(* CODESYS project ET3rdPartyDevices.library
   Version: 3.1.0.4
   Placeholder: ETX
   Description: Engineering Toolbox Extension Library for 3rd party devices
      
      The library is provided "as-is" for TwinCAT3.1 by the Beckhoff Industry Management for Electronics Manufacturing.
      The use of the Library is at the Customer's own risk
      Please check the "DisclaimerStatement" function of the EngineeringToolbox library >= v3.1.0.0
   Title: EngineeringToolboxExtension
   DefaultNamespace: ETX
   Company: Beckhoff Electronics Mfg

Project tree, tasks and I/O mapping:
  libraries: EngineeringToolbox, * (Beckhoff Electronics Mfg); Tc2_EtherCAT, * (Beckhoff Automation GmbH); Tc2_Standard, * (Beckhoff Automation GmbH); Tc2_System, * (Beckhoff Automation GmbH); Tc2_Utilities, * (Beckhoff Automation GmbH); Tc3_Module, * (Beckhoff Automation GmbH)
  GVLs/
  POUs/
    IO/
      Actuators/
        FreqConv/
          EtherCAT/
            DS402/
              Danfoss/
                function block CiA_DS402Controlword_Danfoss [ST]: createControlword
                function block CiA_DS402Statusword_Danfoss [ST]: readStatusword
                function block EcFcDS402_DanfossVLT302 [ST]: setDisable, setEnable, startForward, startReverse, switchOn, forwardStarted, isDisabled, isEnabled, isOff, isOn, reverseStarted
              Lenze/
                function block CiA_DS402Controlword_Lenze [ST]: createControlword
                function block CiA_DS402Statusword_Lenze [ST]: readStatusword
                function block EcFcDS402_LenzeI550 [ST]: setDisable, setEnable, startForward, startReverse, switchOn, forwardStarted, isDisabled, isEnabled, isOff, isOn, reverseStarted
              Parker/
                function block CiA_DS402Controlword_Parker [ST]: createControlword
                function block CiA_DS402Statusword_Parker [ST]: readStatusword
                function block EcFcDS402_ParkerAC30 [ST]: setDisable, setEnable, startForward, startReverse, switchOn, forwardStarted, isDisabled, isEnabled, isOff, isOn, reverseStarted
              Vacon/
                function block CiA_DS402Controlword_Vacon [ST]: createControlword
                function block CiA_DS402Statusword_Vacon [ST]: readStatusword
                function block EcFcDS402_VaconInd100 [ST]: setDisable, setEnable, startForward, startReverse, switchOn, forwardStarted, isDisabled, isEnabled, isOff, isOn, reverseStarted
            function block EcFcComSEW [ST]: reset, setContactorOFF, setContactorON, startBackward, startForward, switchOff, switchOn, backwardStarted, forwardStarted, inError, isBusy, isOff, isOn, noFeed, ok
        function block BlockEconomySmart [ST]: baseClock, reset
      Drives/
        CoE/
          InovanceSV660/
            function block AxDriveCoE_INOVNACE_wEvents [ST]
            function block CiA_DS402Statusword_INOVANCE [ST]: readStatusword
          StaeubliCS8/
            function block AxDriveCoE_StaeubliCS8 [ST]: confirm
            function block CiA_DS402Statusword_StaeubliCS8 [ST]: readStatusword
  VISUs/
*)

// POUs/IO/Actuators/FreqConv/EtherCAT/DS402/Danfoss/CiA_DS402Controlword_Danfoss
FUNCTION_BLOCK CiA_DS402Controlword_Danfoss EXTENDS CiA_DS402Controlword
VAR_INPUT
	EnableRamp						: BOOL; //Operation mode specific Bit 4 -> False = Quick stop / Switch on disabled  
	RunEnable						: BOOL;(* Operation mode specific Bit 5, False = Freeze, the given output frequency is maintained even iF the reference is changed. 
												TRUE = the frequency converter is again able to regulate, and the given reference is followed  *)
	Start							: BOOL;	(* Operation mode specific BIT 6 -> TRUE = gives a start command to the frequency converter / FALSE = the frequency converter controls the motor down to stop  *)

	Jog1On							: BOOL; //	Manufacturere specific Bit 11 Activation of pre-programmed speed in 8-90 Bus Jog 1 Speed JOG 1 is only possible if Bit 04="0", and bit 00-03="1". 

	SetupSelectLSB					: BOOL; //	Manufacturere specific Bit 13
		
	SetupSelectMSB					: BOOL; //	Manufacturere specific Bit 14
	Reversing						: BOOL; // Manufacturere specific Bit 15 
END_VAR
VAR_OUTPUT
END_VAR
VAR
END_VAR

;

METHOD PUBLIC createControlword : UINT
VAR_INPUT
	StatusState												: eCiA_DS402_STATUS_STATE;
END_VAR
	
	createControlword										:= SUPER^.createControlword(StatusState);
	createControlword.4										:= EnableRamp;
	createControlword.5										:= RunEnable;	
	createControlword.6										:= Start;	
	createControlword.11									:= Jog1On;	
	createControlword.13									:= SetupSelectLSB;	
	createControlword.14									:= SetupSelectMSB;	
	createControlword.15									:= Reversing;		
	
				
(*****************************************************************************)
END_METHOD

END_FUNCTION_BLOCK

// POUs/IO/Actuators/FreqConv/EtherCAT/DS402/Danfoss/CiA_DS402Statusword_Danfoss
FUNCTION_BLOCK CiA_DS402Statusword_Danfoss EXTENDS CiA_DS402Statusword
VAR_INPUT
END_VAR
VAR_OUTPUT	
	TargetReached				: BOOL; // Bit 10 in Velocity
	Running						: BOOL; //Bit 14
END_VAR

METHOD PUBLIC readStatusword : BOOL
VAR_INPUT
	Statusword 					:	UINT;
END_VAR


	TargetReached											:= Statusword.10;
	Running													:= Statusword.14;

	readStatusword											:= SUPER^.readStatusword(Statusword);
END_METHOD

END_FUNCTION_BLOCK

// POUs/IO/Actuators/FreqConv/EtherCAT/DS402/Danfoss/EcFcDS402_DanfossVLT302
{attribute 'no_check'}
// Control Danfoss frequency converter in FC mode
FUNCTION_BLOCK EcFcDS402_DanfossVLT302 EXTENDS EcFcDS402_ComBase IMPLEMENTS I_ActuatorFwdRev
VAR_INPUT
	VeloReference											: 	LREAL := 0.0;  	//[RPM] reference velocity
	RampUp													:	LREAL := 1.0;	//[s] sets slope of ramp
	RampDown												:	LREAL := 1.0;	//[s] sets slope of ramp
 
END_VAR                     							
VAR_OUTPUT                  							
	CiA_Control												:	CiA_DS402Controlword_Danfoss;
	CiA_Status												:	CiA_DS402Statusword_Danfoss;
	ErrorCode										AT  %I*	:	UDINT; 			//1690: see also Danfoss documentation
	OpHours											AT  %I* : 	UDINT;			//1500: Operating Hours
	ActPower												: 	LREAL;			//actual scaled Power of drive 
	ActVelo													: 	LREAL;			//actual scaled velocity of drive
	ActCurrent												: 	LREAL;			//actual current consumption of drive
	Q_TargetVelo									AT  %Q* : 	INT;			//1682: Frequence converter set value velocity
	Q_RampUp										AT  %Q* :	UDINT;			// 341: Frequence converter ramp time up
	Q_RampDown										AT  %Q* :	UDINT;			// 342: Frequence converter ramp time down 
END_VAR                 							
VAR (* IO Internal *)   							
                        							
	_ActVelo										AT  %I* : 	INT; 			//1605: Frequence converter actual velocity in digits based on VeloReference
	_ActCurrent										AT  %I* : 	DINT;			//1614: actual current consumption of drive
	_Power											AT  %I* : 	DINT;			//1610: Power 
END_VAR                 								
VAR                     	
END_VAR

(* Com Danfoss VLT302 over Ethercat Gateway MCA 124 	V1.0	 	*)
// ******************************************************************
{info 'FB EcFcDS402_DanfossVLT302: set parameter 4-10 to [2] both directions'}

(* Protection Switch *******************************************)		
	IF ResetTrig  
	THEN 
		REset(); 
	END_IF
	
	ProtSwitchOK();	
	FuseBreakOK(); (* same parameter like ProtSwitch *)

(* Contactor ***************************************************)
	Q_Contactor 											:= Contactor AND ProtSwitchOK.Q AND FuseBreakOK.Q;

(* Read status *************************************************)
	CiA_Status.readStatusword(Statusword);

(* interpret status word ***************************************)
	ActVelo													:= SCALE(_ActVelo, -16384, 16384, -VeloReference, VeloReference);	//16#F000 = -16384 | 16#4000 = 16384    
	ActCurrent             									:= TO_LREAL(_ActCurrent) / 100.0;
	ActPower												:= TO_LREAL(_Power) / 100.0;
	
	Ready													:= CiA_Status.ReadyToSwitchOn AND Q_Contactor;
	Error													:= CiA_Status.Fault AND Q_Contactor;                       									
	Busy													:= CiA_Status.OperationEnabled AND ActVelo <> 0; 
	                                        
// write contorlword DS 402  ****************************************
	CiA_Control.SwitchOn									:= Enable AND Q_Contactor;
	CiA_Control.EnableOperation								:= FeedBwd AND StartBwd AND NOT Start OR Feed AND Start AND NOT StartBwd;
	CiA_Control.FaultReset									:= ResetIntern;
	
	CiA_Control.EnableRamp			 						:= TRUE;
	CiA_Control.RunEnable									:= CiA_Control.SwitchOn;							       
	CiA_Control.Start										:= CiA_Control.EnableOperation;						                     	
	CiA_Control.Reversing			 						:= Start AND NOT StartBwd;	// 15 Reverse     
			
(* setvalue ***************************************************)
	IF CiA_Control.EnableOperation
	THEN
		Q_TargetVelo										:= TO_INT(SCALE(Velo, 	0, VeloReference, 0, 16384));
	ELSE
		Q_TargetVelo										:= 0;
	END_IF
	
	Q_RampUp 												:= TO_UDINT(RampUp*100);
	Q_RampDown 												:= TO_UDINT(RampDown*100);
	              
// Reset FALSE ****************************************************
	ResetIntern												:= FALSE;
	
(* HmiStatus **************************************************)
	Status.0 												:= CiA_Status.OperationEnabled AND StartBwd; 	// counter-clockwise rotation
	Status.1 												:= CiA_Status.OperationEnabled AND Start; 	// clockwise rotation
	Status.2 												:= ActVelo < 0;
	Status.3												:= ActVelo > 0;
	Status.4 												:= FeedBwd;
	Status.5 												:= Feed;
	Status.6 												:= Ready;
	Status.7 												:= Error;
// ****************************************************************

METHOD setDisable : BOOL
VAR_INPUT
END_VAR

SetDisable													:= Super^.setDisable() AND NOT CiA_Status.SwitchedOn;
END_METHOD

METHOD setEnable : BOOL
VAR_INPUT
END_VAR

SetEnable													:= SUPER^.setEnable() AND CiA_Status.SwitchedOn;
END_METHOD

METHOD PUBLIC startForward : bool //Return busy flag
VAR_INPUT
END_VAR
Start 														:= TRUE; 
StartBwd 													:= FALSE;
startForward												:= Busy and Q_TargetVelo > 0;
END_METHOD

METHOD PUBLIC startReverse : bool //Return busy flag
VAR_INPUT
END_VAR
Start 														:= FALSE; 
StartBwd 													:= TRUE;
startReverse												:= Busy and Q_TargetVelo < 0;
END_METHOD

METHOD PUBLIC switchOn : BOOL  //True if motor is switched on
VAR_INPUT
END_VAR
switchOn := startForward();
END_METHOD

{attribute 'monitoring' := 'call'}
PROPERTY public forwardStarted : BOOL
GET
forwardStarted := CiA_Control.EnableOperation and Q_TargetVelo > 0;
END_GET
END_PROPERTY

{attribute 'monitoring' := 'call'}
PROPERTY public isDisabled : BOOL
GET
isDisabled := not CiA_Status.SwitchedOn and not CiA_Status.OperationEnabled;
END_GET
END_PROPERTY

{attribute 'monitoring' := 'call'}
PROPERTY public isEnabled : BOOL
GET
isEnabled := CiA_Status.SwitchedOn or CiA_Status.OperationEnabled;
END_GET
END_PROPERTY

{attribute 'monitoring' := 'call'}
PROPERTY public isOff : BOOL
GET
isOff := NOT CiA_Status.OperationEnabled;
END_GET
END_PROPERTY

{attribute 'monitoring' := 'call'}
PROPERTY public isOn : BOOL
GET
isOn := CiA_Status.OperationEnabled;
END_GET
END_PROPERTY

{attribute 'monitoring' := 'call'}
PROPERTY public reverseStarted : BOOL
GET
reverseStarted := CiA_Control.EnableOperation and Q_TargetVelo < 0;
END_GET
END_PROPERTY

END_FUNCTION_BLOCK

// POUs/IO/Actuators/FreqConv/EtherCAT/DS402/Lenze/CiA_DS402Controlword_Lenze
FUNCTION_BLOCK CiA_DS402Controlword_Lenze EXTENDS CiA_DS402Controlword
VAR_INPUT
	Halt 					: BOOL; // Manufacturere specific Bit 8 - TRUE = stop motor
	ReleaseBreak			: BOOL; //Manufacturere specific Bit 14 
END_VAR
VAR_OUTPUT
END_VAR
VAR
END_VAR

;

METHOD PUBLIC createControlword : UINT
VAR_INPUT
	StatusState												: eCiA_DS402_STATUS_STATE;
END_VAR
	
	createControlword										:= SUPER^.createControlword(StatusState);
	createControlword.8										:= Halt;
	createControlword.8										:= ReleaseBreak;	
	
(*****************************************************************************)
END_METHOD

END_FUNCTION_BLOCK

// POUs/IO/Actuators/FreqConv/EtherCAT/DS402/Lenze/CiA_DS402Statusword_Lenze
FUNCTION_BLOCK CiA_DS402Statusword_Lenze EXTENDS CiA_DS402Statusword
VAR_INPUT
END_VAR
VAR_OUTPUT	
	RPDOsNotActive				:	 BOOL; //Manufacturer specific_Bit8	

	TargetReached				: BOOL; // Bit 10 in velocity 

	BreakOpened					: BOOL; //Manufacturer specific_Bit14
	StoNotActive				: BOOL; //Manufacturer specific_Bit15
END_VAR

METHOD PUBLIC readStatusword : BOOL
VAR_INPUT
	Statusword 					:	UINT;
END_VAR
	RPDOsNotActive											:= Statusword.8;

	TargetReached											:= Statusword.10;

	BreakOpened												:= Statusword.14;
	StoNotActive											:= Statusword.15;

	readStatusword											:= SUPER^.readStatusword(Statusword);
END_METHOD

END_FUNCTION_BLOCK

// POUs/IO/Actuators/FreqConv/EtherCAT/DS402/Lenze/EcFcDS402_LenzeI550
{attribute 'no_check'}
FUNCTION_BLOCK EcFcDS402_LenzeI550 EXTENDS EcFcDS402_ComBase IMPLEMENTS I_ActuatorFwdRev
VAR_INPUT
END_VAR                     							                 							
VAR_OUTPUT                  								
	ActVelo											AT  %I* : 	INT; 			//Actual velocity in rpm
	CiA_Control										:	CiA_DS402Controlword_Lenze;
	CiA_Status										:	CiA_DS402Statusword_Lenze;
	Q_TargetVelo								AT  %Q* : 	INT; 			//Set velocity in rpm
END_VAR                 							                 							
VAR    		
END_VAR

(* Com Lenze i550 over Ethercat Gateway 							*)
(********************************************************************)

(* Protection Switch *******************************************)		
	IF ResetTrig  
	THEN 
		REset(); 
	END_IF
	
	ProtSwitchOK();	
	FuseBreakOK(); (* same parameter like ProtSwitch *)

(* Contactor ***************************************************)
	Q_Contactor 											:= Contactor AND ProtSwitchOK.Q AND FuseBreakOK.Q;
	
(* Read status *************************************************)
	CiA_Status.readStatusword(Statusword);

(* interpret status word ***************************************)
	Ready													:= CiA_Status.ReadyToSwitchOn AND Q_Contactor;
	Error													:= CiA_Status.Fault AND Q_Contactor;                       									
	Busy													:= CiA_Status.OperationEnabled AND ActVelo <> 0; 
	                        	
(* write contorlword DS 402  **********************************)
	CiA_Control.SwitchOn									:= Enable AND Q_Contactor;
	CiA_Control.EnableOperation								:= FeedBwd AND StartBwd AND NOT Start OR Feed AND Start AND NOT StartBwd;
	CiA_Control.FaultReset									:= ResetIntern;	
	           									
(* setvalue ***************************************************)
	IF CiA_Control.EnableOperation
	THEN
		Q_TargetVelo										:= SEL(StartBwd, TO_INT(Velo), TO_INT(Velo) * -1);
	ELSE
		Q_TargetVelo										:= 0;
	END_IF

(* Write control word ******************************************)
	ControlWord 											:= CiA_Control.createControlword(CiA_Status.State);

(* Ack FALSE ***************************************************)
	ResetIntern												:= FALSE;
	
(* HmiStatus **************************************************)
	Status.0 												:= CiA_Status.OperationEnabled AND StartBwd; 	// counter-clockwise rotation
	Status.1 												:= CiA_Status.OperationEnabled AND Start; 	// clockwise rotation
	Status.2 												:= ActVelo < 0;
	Status.3												:= ActVelo > 0;
	Status.4 												:= FeedBwd;
	Status.5 												:= Feed;
	Status.6 												:= Ready;
	Status.7 												:= Error;
	                    									

(**************************************************************)

METHOD setDisable : BOOL
VAR_INPUT
END_VAR

SetDisable													:= Super^.setDisable() AND NOT CiA_Status.SwitchedOn;
END_METHOD

METHOD setEnable : BOOL
VAR_INPUT
END_VAR

SetEnable													:= SUPER^.setEnable() AND CiA_Status.SwitchedOn;
END_METHOD

METHOD PUBLIC startForward : bool //Return busy flag
VAR_INPUT
END_VAR
Start 														:= TRUE; 
StartBwd 													:= FALSE;
startForward												:= Busy and Q_TargetVelo > 0;
END_METHOD

METHOD PUBLIC startReverse : bool //Return busy flag
VAR_INPUT
END_VAR
Start 														:= FALSE; 
StartBwd 													:= TRUE;
startReverse												:= Busy and Q_TargetVelo < 0;
END_METHOD

METHOD PUBLIC switchOn : BOOL  //True if motor is switched on
VAR_INPUT
END_VAR
switchOn := startForward();
END_METHOD

{attribute 'monitoring' := 'call'}
PROPERTY public forwardStarted : BOOL
GET
forwardStarted := CiA_Control.EnableOperation and Q_TargetVelo > 0;
END_GET
END_PROPERTY

{attribute 'monitoring' := 'call'}
PROPERTY public isDisabled : BOOL
GET
isDisabled := not CiA_Status.SwitchedOn and not CiA_Status.OperationEnabled;
END_GET
END_PROPERTY

{attribute 'monitoring' := 'call'}
PROPERTY public isEnabled : BOOL
GET
isEnabled := CiA_Status.SwitchedOn or CiA_Status.OperationEnabled;
END_GET
END_PROPERTY

{attribute 'monitoring' := 'call'}
PROPERTY public isOff : BOOL
GET
isOff := NOT CiA_Status.OperationEnabled;
END_GET
END_PROPERTY

{attribute 'monitoring' := 'call'}
PROPERTY public isOn : BOOL
GET
isOn := CiA_Status.OperationEnabled;
END_GET
END_PROPERTY

{attribute 'monitoring' := 'call'}
PROPERTY public reverseStarted : BOOL
GET
reverseStarted := CiA_Control.EnableOperation and Q_TargetVelo < 0;
END_GET
END_PROPERTY

END_FUNCTION_BLOCK

// POUs/IO/Actuators/FreqConv/EtherCAT/DS402/Parker/CiA_DS402Controlword_Parker
FUNCTION_BLOCK CiA_DS402Controlword_Parker EXTENDS CiA_DS402Controlword
VAR_INPUT
	EnableRampOutput				: BOOL; //Operation mode specific Bit 4 - =0 to set ramp output to zero
	EnableRamp						: BOOL;	//Operation mode specific Bit 5 - =0 to hold ramp
	EnableRampInput					: BOOL;	//Operation mode specific Bit 6 - =0 to set ramp input to zero

	Jog1On							: BOOL; //	Manufacturere specific Bit 8 	

	AutoInitialise					: BOOL; //	Manufacturere specific Bit 12 - 1 = Allow SWITCH ON DISABLED to READY TO SWITCH ON transition regardless of bit 0 (Switch On)
	EnableRevOp						: BOOL; //	Manufacturere specific Bit 13 - 1 = Run Reverse
	RemoteCtrl						: BOOL; //	Manufacturere specific Bit 14 - 0 = Local Sequencing
	RemoteRef						: BOOL; //	Manufacturere specific Bit 15 - 0 = Local Reference
END_VAR
VAR_OUTPUT
END_VAR
VAR
END_VAR

;

METHOD PUBLIC createControlword : UINT
VAR_INPUT
	StatusState												: eCiA_DS402_STATUS_STATE;
END_VAR
	
	createControlword										:= SUPER^.createControlword(StatusState);
	createControlword.4										:= EnableRampOutput;
	createControlword.5										:= EnableRamp;	
	createControlword.6										:= EnableRampInput;	
	createControlword.12									:= AutoInitialise;	
	createControlword.13									:= EnableRevOp;	
	createControlword.14									:= RemoteCtrl;	
	createControlword.15									:= RemoteRef;		
	
(*****************************************************************************)
END_METHOD

END_FUNCTION_BLOCK

// POUs/IO/Actuators/FreqConv/EtherCAT/DS402/Parker/CiA_DS402Statusword_Parker
FUNCTION_BLOCK CiA_DS402Statusword_Parker EXTENDS CiA_DS402Statusword
VAR_INPUT
END_VAR
VAR_OUTPUT	
	TargetReached				: BOOL; // Bit 10 
	Running						: BOOL; //Bit 14
END_VAR

METHOD PUBLIC readStatusword : BOOL
VAR_INPUT
	Statusword 					:	UINT;
END_VAR


	TargetReached											:= Statusword.10;
	Running													:= Statusword.14;

	readStatusword											:= SUPER^.readStatusword(Statusword);
END_METHOD

END_FUNCTION_BLOCK

// POUs/IO/Actuators/FreqConv/EtherCAT/DS402/Parker/EcFcDS402_ParkerAC30
{attribute 'no_check'}
FUNCTION_BLOCK EcFcDS402_ParkerAC30 EXTENDS EcFcDS402_ComBase IMPLEMENTS I_ActuatorFwdRev
VAR_INPUT
	RefVelo													: 	LREAL := 2000; 	//sets speed of rotation	
	RampUp											AT  %Q*	:	TIME := T#10S;	//0486: Acceleration Time
	RampDown										AT  %Q*	:	TIME := T#10S;	//0487: Deceleration Time
END_VAR                     							
VAR_OUTPUT               
	CiA_Control												:	CiA_DS402Controlword_Parker;
	CiA_Status												:	CiA_DS402Statusword_Parker;

	{attribute 'displaymode':='hex'}   							
	WarningCode										AT  %I*	:	UDINT;			//0829: Warnings  1 - 32
	ActVelo											AT  %I* : 	REAL; 			//0395: Actual Speed Percent
	Power											AT  %I*	: 	REAL; 			//0380: Power kW
	Q_TargetVelo							 	AT  %Q* :	REAL;			//0681: Comms Reference
END_VAR                 							
VAR (* IO Internal *)   							
END_VAR                 								
VAR                     	
END_VAR

(* Com Parker AC30 										V1.0   *)
(***************************************************************)

(* Protection Switch *******************************************)		
	IF ResetTrig  
	THEN 
		REset(); 
	END_IF
	
	ProtSwitchOK();	
	FuseBreakOK(); (* same parameter like ProtSwitch *)

(* Contactor ***************************************************)
	Q_Contactor 											:= Contactor AND ProtSwitchOK.Q AND FuseBreakOK.Q;

(* Read status *************************************************)
	CiA_Status.readStatusword(Statusword);

(* interpret status word ***************************************)
	Ready													:= CiA_Status.ReadyToSwitchOn AND Q_Contactor;
	Error													:= CiA_Status.Fault AND Q_Contactor;                       									
	Busy													:= CiA_Status.OperationEnabled AND ActVelo <> 0; 
	                                        
// write contorlword DS 402  ****************************************
	CiA_Control.SwitchOn									:= Enable AND Q_Contactor;
	CiA_Control.EnableOperation								:= FeedBwd AND StartBwd AND NOT Start OR Feed AND Start AND NOT StartBwd;
	CiA_Control.FaultReset									:= ResetIntern;
	CiA_Control.EnableRevOp									:= CiA_Control.EnableOperation AND 	StartBwd;						

(* setvalue ***************************************************)
	IF CiA_Control.EnableOperation AND RefVelo <> 0.0
	THEN
		IF StartBwd
		THEN
			Q_TargetVelo 									:= TO_REAL(Velo/RefVelo * 100.0  * -1); (* 1 Digit = 1 rpm *)
		ELSE	
			Q_TargetVelo									:= TO_REAL(Velo/RefVelo * 100.0); (* 1 Digit = 1 rpm *)
		END_IF	
	ELSE
		Q_TargetVelo										:= 0;
	END_IF
	
// Reset FALSE ****************************************************
	ResetIntern												:= FALSE;
	
(* HmiStatus **************************************************)
	Status.0 												:= CiA_Status.OperationEnabled AND StartBwd; 	// counter-clockwise rotation
	Status.1 												:= CiA_Status.OperationEnabled AND Start; 	// clockwise rotation
	Status.2 												:= ActVelo < 0;
	Status.3												:= ActVelo > 0;
	Status.4 												:= FeedBwd;
	Status.5 												:= Feed;
	Status.6 												:= Ready;
	Status.7 												:= Error;
// ****************************************************************

METHOD setDisable : BOOL
VAR_INPUT
END_VAR

SetDisable													:= Super^.setDisable() AND NOT CiA_Status.SwitchedOn;
END_METHOD

METHOD setEnable : BOOL
VAR_INPUT
END_VAR

SetEnable													:= SUPER^.setEnable() AND CiA_Status.SwitchedOn;
END_METHOD

METHOD PUBLIC startForward : bool //Return busy flag
VAR_INPUT
END_VAR
Start 														:= TRUE; 
StartBwd 													:= FALSE;
startForward												:= Busy and Q_TargetVelo > 0;
END_METHOD

METHOD PUBLIC startReverse : bool //Return busy flag
VAR_INPUT
END_VAR
Start 														:= FALSE; 
StartBwd 													:= TRUE;
startReverse												:= Busy and Q_TargetVelo < 0;
END_METHOD

METHOD PUBLIC switchOn : BOOL  //True if motor is switched on
VAR_INPUT
END_VAR
switchOn := startForward();
END_METHOD

{attribute 'monitoring' := 'call'}
PROPERTY public forwardStarted : BOOL
GET
forwardStarted := CiA_Control.EnableOperation and Q_TargetVelo > 0;
END_GET
END_PROPERTY

{attribute 'monitoring' := 'call'}
PROPERTY public isDisabled : BOOL
GET
isDisabled := not CiA_Status.SwitchedOn and not CiA_Status.OperationEnabled;
END_GET
END_PROPERTY

{attribute 'monitoring' := 'call'}
PROPERTY public isEnabled : BOOL
GET
isEnabled := CiA_Status.SwitchedOn or CiA_Status.OperationEnabled;
END_GET
END_PROPERTY

{attribute 'monitoring' := 'call'}
PROPERTY public isOff : BOOL
GET
isOff := NOT CiA_Status.OperationEnabled;
END_GET
END_PROPERTY

{attribute 'monitoring' := 'call'}
PROPERTY public isOn : BOOL
GET
isOn := CiA_Status.OperationEnabled;
END_GET
END_PROPERTY

{attribute 'monitoring' := 'call'}
PROPERTY public reverseStarted : BOOL
GET
reverseStarted := CiA_Control.EnableOperation and Q_TargetVelo < 0;
END_GET
END_PROPERTY

END_FUNCTION_BLOCK

// POUs/IO/Actuators/FreqConv/EtherCAT/DS402/Vacon/CiA_DS402Controlword_Vacon
FUNCTION_BLOCK CiA_DS402Controlword_Vacon EXTENDS CiA_DS402Controlword
VAR_INPUT
	AlarmReset				:	BOOL; //Manufacturere specific Bit 12 

END_VAR
VAR_OUTPUT
END_VAR
VAR
END_VAR

;

METHOD PUBLIC createControlword : UINT
VAR_INPUT
	StatusState												: eCiA_DS402_STATUS_STATE;
END_VAR
	
	createControlword										:= SUPER^.createControlword(StatusState);
	createControlword.11									:= AlarmReset;	
	
(*****************************************************************************)
END_METHOD

END_FUNCTION_BLOCK

// POUs/IO/Actuators/FreqConv/EtherCAT/DS402/Vacon/CiA_DS402Statusword_Vacon
FUNCTION_BLOCK CiA_DS402Statusword_Vacon EXTENDS CiA_DS402Statusword
VAR_INPUT
END_VAR
VAR_OUTPUT	
	TargetReached				: BOOL; // Bit 10 commonly used FOR in target position, velocity ect.
	IncorrectDriveMode		:	BOOL; //Manufacturer specific_Bit14
END_VAR

METHOD PUBLIC readStatusword : BOOL
VAR_INPUT
	Statusword 					:	UINT;
END_VAR


	TargetReached											:= Statusword.10;

	IncorrectDriveMode										:= Statusword.14;


	readStatusword											:= SUPER^.readStatusword(Statusword);
END_METHOD

END_FUNCTION_BLOCK

// POUs/IO/Actuators/FreqConv/EtherCAT/DS402/Vacon/EcFcDS402_VaconInd100
{attribute 'no_check'}
FUNCTION_BLOCK EcFcDS402_VaconInd100 EXTENDS EcFcDS402_ComBase IMPLEMENTS I_ActuatorFwdRev
VAR_INPUT
END_VAR                     							
VAR_OUTPUT                  								
	CiA_Control										:	CiA_DS402Controlword_Vacon;
	CiA_Status										:	CiA_DS402Statusword_Vacon;
	_1_OutputFreq 							AT  %I*	:	UINT; // 0,01 Hz
	_2_Act_rpm								AT  %I*	:	UINT; // 1/MIN
	_3_ActCurrent							AT  %I*	:	UINT; // 0,1 A
	_4_ActTorque							AT  %I*	:	UINT; // 0.1%
	_5_ActPower								AT  %I*	:	UINT; // 0.1%
	_6_ActVoltage							AT  %I*	:	UINT; // 0,1 V
	_7_DClinkVoltage						AT  %I*	:	UINT; // 1 V
	_8_LastErrorCode						AT  %I*	:	UINT; //  
	Q_TargetVelo									AT  %Q* : 	INT; 			//Set velocity in rpm
END_VAR                 							
VAR (* IO Internal *)   							

END_VAR

(* Com Vacon 100 +SDEC EtherCAT Fieldbus option Board 	V1.0   *)
(***************************************************************)
																													
(* Protection Switch *******************************************)		
	IF ResetTrig  
	THEN 
		REset(); 
	END_IF
	
	ProtSwitchOK();	
	FuseBreakOK(); (* same parameter like ProtSwitch *)

(* Contactor ***************************************************)
	Q_Contactor 											:= Contactor AND ProtSwitchOK.Q AND FuseBreakOK.Q;
	
(* Read status *************************************************)
	CiA_Status.readStatusword(Statusword);

(* interpret status word ***************************************)
	Ready													:= CiA_Status.ReadyToSwitchOn AND Q_Contactor;
	Error													:= CiA_Status.Fault AND Q_Contactor;                       									
	Busy													:= CiA_Status.OperationEnabled AND _2_Act_rpm <> 0; 
	                        	
(* write contorlword DS 402  **********************************)
	CiA_Control.SwitchOn									:= Enable AND Q_Contactor;
	CiA_Control.EnableOperation								:= FeedBwd AND StartBwd AND NOT Start OR Feed AND Start AND NOT StartBwd;
	CiA_Control.FaultReset									:= ResetIntern;	
	CiA_Control.AlarmReset									:= ResetIntern;	
	           									
(* setvalue ***************************************************)
	IF CiA_Control.EnableOperation
	THEN
		Q_TargetVelo										:= SEL(StartBwd, TO_INT(Velo), TO_INT(Velo) * -1);
	ELSE
		Q_TargetVelo										:= 0;
	END_IF

(* Write control word ******************************************)
	ControlWord 											:= CiA_Control.createControlword(CiA_Status.State);

(* Ack FALSE ***************************************************)
	ResetIntern												:= FALSE;
	
(* HmiStatus **************************************************)
	Status.0 												:= CiA_Status.OperationEnabled AND StartBwd; 	// counter-clockwise rotation
	Status.1 												:= CiA_Status.OperationEnabled AND Start; 	// clockwise rotation
	Status.2 												:= _2_Act_rpm < 0;
	Status.3												:= _2_Act_rpm > 0;
	Status.4 												:= FeedBwd;
	Status.5 												:= Feed;
	Status.6 												:= Ready;
	Status.7 												:= Error;
	                    									

(**************************************************************)

METHOD setDisable : BOOL
VAR_INPUT
END_VAR

SetDisable													:= Super^.setDisable() AND NOT CiA_Status.SwitchedOn;
END_METHOD

METHOD setEnable : BOOL
VAR_INPUT
END_VAR

SetEnable													:= SUPER^.setEnable() AND CiA_Status.SwitchedOn;
END_METHOD

METHOD PUBLIC startForward : bool //Return busy flag
VAR_INPUT
END_VAR
Start 														:= TRUE; 
StartBwd 													:= FALSE;
startForward												:= Busy and Q_TargetVelo > 0;
END_METHOD

METHOD PUBLIC startReverse : bool //Return busy flag
VAR_INPUT
END_VAR
Start 														:= FALSE; 
StartBwd 													:= TRUE;
startReverse												:= Busy and Q_TargetVelo < 0;
END_METHOD

METHOD PUBLIC switchOn : BOOL  //True if motor is switched on
VAR_INPUT
END_VAR
switchOn := startForward();
END_METHOD

{attribute 'monitoring' := 'call'}
PROPERTY public forwardStarted : BOOL
GET
forwardStarted := CiA_Control.EnableOperation and Q_TargetVelo > 0;
END_GET
END_PROPERTY

{attribute 'monitoring' := 'call'}
PROPERTY public isDisabled : BOOL
GET
isDisabled := not CiA_Status.SwitchedOn and not CiA_Status.OperationEnabled;
END_GET
END_PROPERTY

{attribute 'monitoring' := 'call'}
PROPERTY public isEnabled : BOOL
GET
isEnabled := CiA_Status.SwitchedOn or CiA_Status.OperationEnabled;
END_GET
END_PROPERTY

{attribute 'monitoring' := 'call'}
PROPERTY public isOff : BOOL
GET
isOff := NOT CiA_Status.OperationEnabled;
END_GET
END_PROPERTY

{attribute 'monitoring' := 'call'}
PROPERTY public isOn : BOOL
GET
isOn := CiA_Status.OperationEnabled;
END_GET
END_PROPERTY

{attribute 'monitoring' := 'call'}
PROPERTY public reverseStarted : BOOL
GET
reverseStarted := CiA_Control.EnableOperation and Q_TargetVelo < 0;
END_GET
END_PROPERTY

END_FUNCTION_BLOCK

// POUs/IO/Actuators/FreqConv/EtherCAT/EcFcComSEW
{attribute 'no_check'}
FUNCTION_BLOCK EcFcComSEW IMPLEMENTS I_ActuatorFwdBwd(* SEW *)
VAR_INPUT
	ResetTrig												:	BOOL := TRUE;	//Resets error with rising edge 
	Start													:	BOOL := FALSE;	//motor rotates in right direction when TRUE
	StartBwd												:	BOOL := FALSE; 	//motor rotates in left direction when TRUE
	Contactor												:	BOOL := FALSE;	//if available
	Enable													:	BOOL := FALSE;	//enables drive
	Feed													:	BOOL := TRUE;	//enables feed in right direction and should be set to FALSE when right limit sensor is reached
	FeedBwd													:	BOOL := TRUE;	//enables feed in left direction and should be set to FALSE when left limit sensor is reached
	Velo													: 	LREAL := 0.0;  	//sets speed of rotation
	Ramp													:	LREAL := 1.0;	//sets slope of ramp
	ProtSwitchOK											: 	FUSE;			//monitors feeding protective device
	FuseBreakOK												: 	FUSE;			//monitors feeding circuit breaker 
END_VAR                     							
VAR_OUTPUT                  							
{attribute 'displaymode':='binary'}
	Status													:	BYTE; 			//for HMI
{attribute 'displaymode':='binary'}
	UnitStatus												:	BYTE; 			(* device status
																				0x0 not ready
																				0x1 controller locked
																				0x2 not enabled
																				0x3 standstill current acitve, not enabled
																				0x4 enabled
																				0x8 default factory settings active *)
	ErrorCode												:	BYTE; 			//see also SEW-documentation
{attribute 'displaymode':='hex'}
	Statusword1										AT  %I* : 	INT;			//status word 1 contains state of drive
	ActVelo													: 	LREAL;			//actual scaled velocity of drive
	ActCurrent										AT  %I* : 	INT;			//actual current consumption of drive
	Ready													:	BOOL;			//TRUE when drive is ready to operate
	Warning													:	BOOL;			//TRUE when a warning is active 
	Busy													:	BOOL;			//Busy is TRUE at the rising edge of Enable and stays TRUE as long as the FB is performing any action. 	
	Error													:	BOOL;			//Rising edge of Error informs that an error occurred during the execution of the Function Block 	 	
END_VAR                 							
VAR (* IO Internal *)
{attribute 'displaymode':='hex'}   							
	Q_Controlword1									AT  %Q* : 	INT;			//Frequence converter controlword 1
	Q_TargetVelo									AT  %Q* : 	INT;			//Frequence converter set target velocity in digits
	Q_Ramp											AT  %Q* :	INT;			//Frequence converter ramp time in 
                        							
	Q_Contactor 									AT  %Q* :	BOOL;			//Hardware output 
	_ActVeloDigit									AT  %I* : 	INT; 			//Frequence converter actual velocity in digits based on rpm 
END_VAR                 								
VAR    
	QuitIntern												:	BOOL;                 	
END_VAR

(* Com SEW MovitracB over Ethercat Gateway 		V2.0	*)
(********************************************************)

(* Protection Switch *****************************************)
	IF ResetTrig 
	THEN 
		reset(); 
	END_IF
	
	ProtSwitchOK();
	FuseBreakOK(); (* same parameter like ProtSwitch *)

(* Contactor ********************************************************)
	Q_Contactor 											:= Contactor AND ProtSwitchOK.Q AND FuseBreakOK.Q;

(* interpret status word *********************************)
	(*EndstufeFRG											:= Statusword1.0; *)
	Ready													:= Statusword1.1 AND Q_Contactor;
	Warning													:= Statusword1.5 AND Ready ;
	Error													:= Statusword1.5 AND NOT Ready AND Q_Contactor ;
	(*EndlLinksAktiv 										:= Statusword1.6; *)
	(*EndlLinksAktiv 										:= Statusword1.7; *)
                        									
	ActVelo													:= INT_TO_LREAL(_ActVeloDigit) * 0.2;
	Busy													:= Ready AND Q_Controlword1.2 AND ActVelo > 5.0;
                        	
(* interpret HighByte status word 1 ********************)
	(* Init *)
	UnitStatus := ErrorCode 								:= 0;

	IF Q_Contactor THEN
		IF NOT Statusword1.5 THEN
			UnitStatus.0 									:= Statusword1.8;
			UnitStatus.1 									:= Statusword1.9;
			UnitStatus.2 									:= Statusword1.10;
			UnitStatus.3									:= Statusword1.11;
			UnitStatus.4 									:= Statusword1.12;
			UnitStatus.5 									:= Statusword1.13;
			UnitStatus.6 									:= Statusword1.14;
			UnitStatus.7 									:= Statusword1.15;
		ELSE                								
			ErrorCode.0 									:= Statusword1.8;
			ErrorCode.1 									:= Statusword1.9;
			ErrorCode.2 									:= Statusword1.10;
			ErrorCode.3										:= Statusword1.11;
			ErrorCode.4 									:= Statusword1.12;
			ErrorCode.5 									:= Statusword1.13;
			ErrorCode.6 									:= Statusword1.14;
			ErrorCode.7 									:= Statusword1.15;
		END_IF
	END_IF

(* write contorlword 1  *********************************)
	Q_Controlword1.0 										:= FALSE; (* controller locked=1/0=enabled *)
	Q_Controlword1.1 										:= Enable AND Q_Contactor; (* controller enabled=1/0=rapid stop *)
	Q_Controlword1.2 										:= FeedBwd AND StartBwd AND NOT Start
																OR Feed AND Start AND NOT StartBwd; (* enable start FU *)
	Q_Controlword1.6 										:= QuitIntern;
	Q_Controlword1.8 										:= NOT Start AND StartBwd; (* rotation direction 0=right/1=left *)
                        									
(* setvalue **************************************)
	IF 	Start 
		AND NOT StartBwd 
		AND Feed 
	THEN
		Q_TargetVelo 										:= LREAL_TO_INT(Velo) * 5; (* 5 Digit = 1 rpm *)
	ELSIF StartBwd 
		AND NOT Start 
		AND FeedBwd 
	THEN
		Q_TargetVelo 										:= (LREAL_TO_INT(Velo) * 5 ) * -1; (* 5 Digit = 1 rpm *)
	ELSE
		Q_TargetVelo 										:= 0;
	END_IF

(* set ramp ******************************************)
	Q_Ramp	 												:= LREAL_TO_INT(Ramp);

(* Ack FALSE **********************************************)
	QuitIntern												:= FALSE;
	
(* HmiStatus **************************************************)
	Status.0 												:= Q_Controlword1.2 AND Q_Controlword1.8 ; //counter-clockwise rotation
	Status.1 												:= Q_Controlword1.2 AND NOT  Q_Controlword1.8; //clockwise rotation
	Status.2 												:= FALSE;
	Status.3												:= FALSE;
	Status.4 												:= FeedBwd;
	Status.5 												:= Feed;
	Status.7 												:= Ready;
	Status.7 												:= Error;
	                    									

(**************************************************************)

METHOD PUBLIC reset : booL
VAR_INPUT
END_VAR
QuitIntern 	:= Q_Controlword1.6   							:= TRUE;
ProtSwitchOK.reset();
FuseBreakOK.reset();
reset													:= TRUE;
END_METHOD

METHOD PUBLIC setContactorOFF : BOOL //Return true if contactor is off and not busy
VAR_INPUT
END_VAR
Q_Contactor := Contactor 									:=FALSE;
							
SetContactorOFF 											:= TRUE;
END_METHOD

METHOD PUBLIC setContactorON : bool //return true if contactor on
VAR_INPUT
END_VAR
Q_Contactor := Contactor 									:= ProtSwitchOK.Q AND FuseBreakOK.Q ;
SetContactorON												:= Q_Contactor;
END_METHOD

METHOD PUBLIC startBackward : bool //Return busy flag
VAR_INPUT
END_VAR
Start 														:= FALSE; 
StartBwd 													:= TRUE;
Q_Controlword1.2 											:= FeedBwd AND ProtSwitchOK.Q; (* FRG Start FU *)
Q_Controlword1.8 											:= Q_Controlword1.2 ; (* Drehrichtung 0=Rechts/1=Links *)
Busy														:= Q_Controlword1.2;
startBackward												:= Busy;
END_METHOD

METHOD PUBLIC startForward : bool //Return busy flag
VAR_INPUT
END_VAR
Start 														:= TRUE; 
StartBwd 													:= FALSE;
Q_Controlword1.2 											:= Feed AND Start AND NOT StartBwd AND ProtSwitchOK.Q; (* FRG Start FU *)
Q_Controlword1.8 											:= FALSE ; (* Drehrichtung 0=Rechts/1=Links *)
Busy														:= Q_Controlword1.2;
startForward												:= Busy;
END_METHOD

METHOD PUBLIC switchOff : BOOL //Return true if stopped / busy = false
VAR_INPUT
END_VAR
Start 														:= FALSE;
StartBwd													:= FALSE;
Q_Controlword1.2 											:= FALSE;
switchOff													:= NOT Busy;
END_METHOD

METHOD PUBLIC switchOn : BOOL  //True if motor is switched on
VAR_INPUT
END_VAR
switchOn := startForward();
END_METHOD

{attribute 'monitoring' := 'call'}
PROPERTY public backwardStarted : BOOL
GET
backwardStarted := Q_Controlword1.2 and Q_TargetVelo < 0;
END_GET
END_PROPERTY

{attribute 'monitoring' := 'call'}
PROPERTY public forwardStarted : BOOL
GET
forwardStarted := Q_Controlword1.2 and Q_TargetVelo > 0;
END_GET
END_PROPERTY

{attribute 'monitoring' := 'call'}
PROPERTY public inError : bool
GET
inError := Error or not ProtSwitchOK.Q or not FuseBreakOK.Q;
END_GET
END_PROPERTY

{attribute 'monitoring' := 'call'}
PROPERTY public isBusy : bool
GET
isBusy := Busy;
END_GET
END_PROPERTY

{attribute 'monitoring' := 'call'}
PROPERTY public isOff : BOOL
GET
isOff := NOT Q_Contactor or Q_TargetVelo = 0;
END_GET
END_PROPERTY

{attribute 'monitoring' := 'call'}
PROPERTY public isOn : BOOL
GET
isOn := Q_Contactor and Q_TargetVelo <> 0 and not inError;
END_GET
END_PROPERTY

{attribute 'monitoring' := 'call'}
PROPERTY noFeed : BOOL
GET
noFeed := NOT Feed and not FeedBwd;
END_GET
END_PROPERTY

{attribute 'monitoring' := 'call'}
PROPERTY ok : bool
GET
ok := isOn;
END_GET
END_PROPERTY

END_FUNCTION_BLOCK

// POUs/IO/Actuators/BlockEconomySmart
//Block Economy Smart 
//FB is able to control and read all values from Block Ecomemy Smart Fuse
{attribute 'no_check'}
FUNCTION_BLOCK BlockEconomySmart
VAR CONSTANT 										
	MIN_DATA												: INT := 0;
	MAX_DATA												: INT := 96;
END_VAR
VAR_OUTPUT CONSTANT
	MIN_CHANNEL												: INT := 1;
	MAX_CHANNEL												: INT := 8;
	STATUS_ON												: BYTE := 0;
	STATUS_OFF												: BYTE := 1;
	STATUS_TRIP												: BYTE := 2;
	STATUS_OVERCURRENT										: BYTE := 3;
END_VAR                         							
VAR_INPUT                       							
	Enable													: BOOL := TRUE; //Enable communication 
	Force													: ARRAY[MIN_CHANNEL..MAX_CHANNEL] OF BOOL; 	// 	simulates channel
	Control													: ARRAY[MIN_CHANNEL..MAX_CHANNEL] OF BOOL; 	// 	Enable/Disable channel 
	SetCtrl													: BOOL := FALSE;		// 	Write channel control to output (Econemy Smart Fuse)
	ResetTrig												: BOOL := FALSE;		// 	Reset tripped fuses/channels
	ReadSetValues											: BOOL := FALSE;		// 	Read trip set value of all cannels
	ReadChecksum											: BOOL := FALSE;		// 	Read checksumm
	ExtProtocolSampleingDivider								: UINT := 0;			//  0 = read only short protocol / >0 = read long protocol every n cycles 					
END_VAR
VAR_OUTPUT
	Voltage													: LREAL;					// [V] actual voltage
	Current													: ARRAY[MIN_CHANNEL..MAX_CHANNEL] OF LREAL;	// [A] actual cannel current[1-8]
	Status													: ARRAY[MIN_CHANNEL..MAX_CHANNEL] OF BYTE;	// Fuse status
	FuseTripped												: BOOL := FALSE;		// min 1 Fuse has tripped
	UpdateCycle												: UINT := 0;			// update Cycle counter
	Busy													: BOOL; 				// 
	ErrorCom												: BOOL;					// 				
END_VAR
VAR 
	In												AT%I*	: BOOL;
	Out												AT%Q*	: BOOL;
END_VAR
VAR
//local cache ************************************************************************************
	State													: INT := -1;
	CycleTime												: LREAL; // [ms] Cycle Time of PLC Task
	_BaseClock												: INT := 100; // MIN: 70 MAX: 200
	CurrentCycles											: UDINT;
	CyclePerTick											: UDINT;
	_InternReset											: BOOL;

	BitIdx,RecBits											: INT;
	SendData												: ARRAY[MIN_DATA..MAX_DATA] OF BOOL;
	ReceiveBits												: ARRAY[MIN_DATA..MAX_DATA] OF BOOL;
	ReceiveBytes											: ARRAY[MIN_DATA..MAX_DATA/8] OF BYTE;
	
	{attribute 'displaymode':='binary'}
	Temp 													: BYTE;		


				
//trigger *********************************************************************************
	
//timer ***********************************************************************************
	Delay													: TON;
	
//instances ***********************************************************************************             								
	GETCURTASKINDEX											: GETCURTASKINDEX;


//Dummys ****************************************************************************************
	i,j														: INT;
END_VAR

	(* Block Economy Smart communication 					*)
	(********************************************************)

(* Initiat reset of channel ***********************************************)
	IF ResetTrig THEN reset();	END_IF

(* State machine to read and write data ************************************)
	CASE State OF
	-1: // init
		GETCURTASKINDEX();
		CycleTime 											:= TwinCAT_SystemInfoVarList._TaskInfo[GETCURTASKINDEX.index].CycleTime / 10_000;
		IF CycleTime > 0 THEN           						
			CyclePerTick									:= LREAL_TO_UDINT(_BaseClock / CycleTime);	
			CyclePerTick									:= CyclePerTick + (CyclePerTick MOD 2);
			State											:= 0;
		END_IF                          						
																
	0: // idle          
		IF Enable
		THEN    	   
			Busy											:= TRUE; 						
			FOR i := MIN_CHANNEL TO MAX_CHANNEL DO    									
				SendData[i]									:= Control[9-i];
			END_FOR                 						
			SendData[9]										:= SetCtrl;			    	
			SendData[10]									:= extProtocolSampleingDivider <> 0
																AND(	
																(UpdateCycle MOD extProtocolSampleingDivider) = 0
																OR UpdateCycle = 0)
																OR ReadSetValues;
			SendData[11]									:= ReadSetValues;
			SendData[12]									:= FALSE;
			SendData[13]									:= FALSE;
			SendData[14]									:= ReadChecksum AND NOT SetCtrl;
			BitIdx											:= 0;		
			State											:= SEL(_InternReset, 10, 5); // Reset tripped if flag is true
			RecBits											:= SEL( SendData[10], 16, 88) 	// short / long
															+  SEL( ReadChecksum, 0, 8);	// checksum on/off
		ELSE
			Busy											:= FALSE;
			Out												:= FALSE;
			State											:= 0;
			Voltage											:= 0.0;
			MEMSET(ADR(Current),0,SIZEOF(Current));			
			MEMSET(ADR(Status),0,SIZEOF(Status));	        
			FuseTripped										:= FALSE;
			UpdateCycle										:= 0;		
		END_IF
																
	5:	//reset triped          								
		Out													:= TRUE;
		Delay(IN:= NOT Delay.Q, PT := T#600MS);             
															
		IF Delay.Q THEN             						
			_InternReset									:= FALSE;
			Delay(IN := FALSE);                             
			State 											:= 20;
		END_IF                  							
															
	10: // receive	            							
		Out													:= SendData[BitIdx] XOR CurrentCycles <= CyclePerTick / 2;		
															
		IF CurrentCycles >= CyclePerTick					 
		THEN                            	                
			ReceiveBits[BitIdx]								:= In;
			CurrentCycles									:= 0;
			BitIdx											:= BitIdx + 1;
			IF BitIdx > RecBits
			THEN
				Out											:= FALSE;
				State										:= 20;
			END_IF                  	
		ELSE	                    	
			CurrentCycles									:= CurrentCycles + 1;
		END_IF
		
	20:	 // interpret Channels
		Delay( IN:= NOT Delay.Q AND NOT IN, PT := TO_TIME(_BaseClock*3));
		IF Delay.Q THEN		// stop Bit		
			Delay(IN := FALSE);
			
			// Cannel Status
			FOR i := MIN_CHANNEL TO MAX_CHANNEL DO	
				IF Force[i] THEN
					Status[i]								:= STATUS_ON;				
				ELSIF ReceiveBits[9-i] AND ReceiveBits[17-i] THEN   
					Status[i]								:= STATUS_OVERCURRENT;	
				ELSIF ReceiveBits[9-i] THEN                     
					Status[i]								:= STATUS_ON;
				ELSIF ReceiveBits[17-i] THEN                    
					Status[i]								:= STATUS_TRIP;
				ELSE                                        
					Status[i]								:= STATUS_OFF;
				END_IF                                      
			END_FOR		                                    
		      
			//  interpret Checksum
			FOR i := MIN_DATA TO MAX_DATA/8 DO
				ReceiveBytes[0+i].0 						:= ReceiveBits[8*i+0];
				ReceiveBytes[0+i].1 						:= ReceiveBits[8*i+1];
				ReceiveBytes[0+i].2 						:= ReceiveBits[8*i+2];
				ReceiveBytes[0+i].3 						:= ReceiveBits[8*i+3];
				ReceiveBytes[0+i].4 						:= ReceiveBits[8*i+4];
				ReceiveBytes[0+i].5 						:= ReceiveBits[8*i+5];
				ReceiveBytes[0+i].6 						:= ReceiveBits[8*i+6];
				ReceiveBytes[0+i].7 						:= ReceiveBits[8*i+7];
			END_FOR
			ErrorCom := 	SendData[14]
						AND (	( ReceiveBytes[1] XOR ReceiveBytes[2]) = ReceiveBytes[3] AND BitIdx < 30
							OR 	((ReceiveBytes[1] XOR ReceiveBytes[2] XOR ReceiveBytes[3] XOR ReceiveBytes[4] XOR ReceiveBytes[5] XOR ReceiveBytes[6] XOR
						 		  ReceiveBytes[7] XOR ReceiveBytes[8] XOR ReceiveBytes[9] XOR ReceiveBytes[10] XOR ReceiveBytes[11]) = ReceiveBytes[12] AND BitIdx > 30)
							 );
                                              
			// set collective triped bit                    
			FuseTripped										:= FALSE;
			FOR i := MIN_CHANNEL TO MAX_CHANNEL DO          
				IF Status[i] = STATUS_TRIP THEN             
					FuseTripped								:= TRUE;
					EXIT;
				END_IF
			END_FOR
			
			// interpret extended protoccol
			IF 	SendData[10] 
				OR 	SendData[11] 
			THEN			
				FOR i := MIN_CHANNEL TO MAX_CHANNEL DO // Voltage
					Temp									:= SHL(Temp,1) OR TO_BYTE(ReceiveBits[16+i]);
				END_FOR		  
				Voltage										:= Temp/16.0 + 16;
				FOR j := MIN_CHANNEL TO MAX_CHANNEL DO // Current[1-8]
					FOR i := MIN_CHANNEL TO MAX_CHANNEL DO    // bit shifting
						Temp								:= SHL(Temp,1) OR TO_BYTE(ReceiveBits[24+((j-1)*8)+i]);
					END_FOR		  
					Current[j]								:= Temp/16.0;
				END_FOR
			END_IF          
				
			UpdateCycle 									:= UpdateCycle + 1; 
			State 											:= 0;
		END_IF	
	END_CASE
	
(*****************************************************************)

PROPERTY PUBLIC baseClock : INT // MIN: 70 MAX: 200
GET
BaseClock := _BaseClock;
END_GET
SET
_BaseClock := LIMIT(70, BaseClock, 200);
State := -1;
END_SET
END_PROPERTY

METHOD reset : BOOL //Resetting tripped channel / Return TRUE as lons as FuseTripped = TRUE
VAR_INPUT
END_VAR
_InternReset													:= FuseTripped;
reset															:= TRUE;
END_METHOD

END_FUNCTION_BLOCK

// POUs/IO/Drives/CoE/InovanceSV660/AxDriveCoE_INOVNACE_wEvents
FUNCTION_BLOCK AxDriveCoE_INOVNACE_wEvents  EXTENDS AxDriveBase (* Inovance SV660N EtherCAT drive 
Do enable remote break control the folloing settings are needed

Required process data: 
- 0x1B01, which includes 0x60FE:01 Physical outputs

Required startup list entries: 
- 0x60FE:02 (Bit Mask) = 400000 dec.
- 0x200D:12 (Forced DI/DO setting) = 4 dec (EtherCAT)
- 0x2004:05 (DO Function Selection) = 9 dec (to set DO function back to drive on restart) 

*)
VAR CONSTANT
	PHY_OUTPUT_BRAKE										:	INT := 18;
END_VAR
VAR_INPUT
	EnableEvent												:	BOOL := TRUE;
	ConfirmTrig												:	BOOL := FALSE; (* Reset event *)
	SourceId												:	UDINT := 102200; //CoE Drive default multisource Id + Ax id
	Name													:	STRING(30) := '';
	ErrorLimitPos											:	BOOL := FALSE;
	ErrorLimitNeg											:	BOOL := FALSE;
	BrakeUnlock												:	BOOL := FALSE;
	PhysicalOutputs									AT%Q*	:   UDINT;
END_VAR
VAR_OUTPUT
	BrakeUnlocked											:	BOOL;
	Status													:	CiA_DS402Statusword_INOVANCE;	

	EventStatus												:	DWORD;
	NoOfActiveEvents										:	INT;
	Busy													:	BOOL;
	Error													:	BOOL;
	ErrorId													:	UDINT;
	STOOff													:	BOOL;
	
	ModesOfOperationDisplay							AT %I*	:	SINT;
	DigitalInputs									AT %I*	:	UDINT;
	ErrorCode										AT %I*	:	UINT;
END_VAR
VAR
END_VAR
VAR
(* Function blocks ****************************************************************************)	
	CoEWrite												: FB_EcCoeSdoWriteEx := (tTimeout := DEFAULT_ADS_TIMEOUT);
	Event													: EventHandlingGrp10;
	i														:	INT;
	BrakeState												:	INT;	
	CoESetValue												:	INT;
END_VAR

	(* CoE Drive																		*)
	(************************************************************************************)

		(* CoE Drive																		*)
	(************************************************************************************)

(* abort function-call if the reference is invalid *****************************)
	IF NOT __ISVALIDREF(rAxis) 
	THEN
		Busy												:= NOT Error;
		Fault												:= TRUE;
		SwitchedOn											:= FALSE;
		Ready												:= FALSE;
		Error												:= TRUE;
		ErrorId												:= 16#4B30;
		RETURN;         										
	END_IF

(* Call super class ****************************************************)
	SUPER^(); 
	
(* Read Statusword ********************************************************)	
	IF rAxis.Status.OpMode.SimulationAxis
	THEN
		IF rAxis.PlcToNc.ControlDWord.0
		THEN
			Status.readStatusword(TO_UINT(eCiA_DS402_STATUS_STATE.OPERATION_ENABLED));
		ELSE
			Status.readStatusword(TO_UINT(eCiA_DS402_STATUS_STATE.SWITCHED_ON));	
		END_IF
	ELSE
		Status.readStatusword(Statusword);
	END_IF	
		
(* DriveStatusBits ***********************************************)
	Fault													:= Status.Fault
																OR rAxis.NcToPlc.StateDWord.28 (* DriveDeviceError *)
																OR rAxis.NcToPlc.StateDWord.30; (* IODataInvalid *)
            												
	Ready 													:= NOT Fault
																AND(Status.ReadyToSwitchOn OR Status.SwitchedOn);

	SwitchedOn												:= Status.SwitchedOn AND NOT Fault;

	STOOff													:= DigitalInputs.3;
	
	
(* manual override break ********************************************************)		
	CASE BrakeState OF
	0:								
		IF BrakeUnlock AND NOT rAxis.PlcToNc.ControlDWord.0 XOR BrakeUnlocked 
		THEN
			CoESetValue										:= SEL(BrakeUnlock AND NOT rAxis.PlcToNc.ControlDWord.0, 9, 31);
			CoEWrite(
				bExecute	:=TRUE  , 
				sNetId		:= F_CreateAmsNetId(nIds :=AdsAddr.netId),
				nSlaveAddr	:= AdsAddr.port,
				nIndex		:= 16#2004,
				nSubIndex	:= 16#5,
				pSrcBuf		:=ADR(CoESetValue) , 
				cbBufLen	:=SIZEOF(CoESetValue));	
			Busy											:= TRUE;
			BrakeState										:= BrakeState + 1;
		END_IF
	
	1:
		CoEWrite( bExecute	:=TRUE  , pSrcBuf	:=ADR(CoESetValue),cbBufLen:=SIZEOF(CoESetValue));	

		IF NOT CoEWrite.bBusy
		THEN
			IF CoEWrite.bError	
			THEN
				BrakeState									:= 99;
			ELSE
				BrakeUnlocked								:= CoESetValue = 31; //Control via EtherCAT
				CoEWrite(bExecute :=FALSE);
				BrakeState									:= 0;
			END_IF
		END_IF
		
	99: //Error CoE Write
		Error												:= TRUE;
		ErrorId												:= CoEWrite.nErrId;
		Busy												:= FALSE;		
		IF ConfirmTrig
		THEN
			CoEWrite( bExecute	:=FALSE  , pSrcBuf	:=ADR(CoESetValue),cbBufLen:=SIZEOF(CoESetValue));		
			Error											:= FALSE;
			ErrorId											:= 0;
			BrakeState										:= 0;	
		END_IF
	END_CASE
	
	//Set pysical output 
	PhysicalOutputs.PHY_OUTPUT_BRAKE						:= BrakeUnlocked;

	
(* Set Tc event messages of status word *****************************************************)
	Event.no[1].Flag 										:= NOT Status.ReadyToSwitchOn AND InfoDataState = Tc2_EtherCAT.EC_DEVICE_STATE_OP; 
	Event.no[2].Flag 										:= Status.Fault OR ErrorCode <> 0; IF Event.no[2].Flag THEN Event.no[1].Text1 := CONCAT(', error code:', DWORD_TO_HEXSTR(TO_DWORD(ErrorCode),4,FALSE));END_IF
	Event.no[3].Flag 										:= Status.Warning; 	 			
	Event.no[4].Flag 										:= Status.InternalLimitActive;
	Event.no[5].Flag 										:= Status.SwitchOnDisabled;
//	Event.no[6].Flag 										:= NOT Status.RemoteSwitch AND Status.SwitchedOn;
	Event.no[7].Flag 										:= BrakeUnlock ; 	
	Event.no[8].Flag 										:= ErrorLimitPos AND InfoDataState = Tc2_EtherCAT.EC_DEVICE_STATE_OP;
	Event.no[9].Flag 										:= ErrorLimitNeg AND InfoDataState = Tc2_EtherCAT.EC_DEVICE_STATE_OP;
//	Event.no[10].Flag 										:= ADC drive error
	
(* Check if msg activ and init some parameter ***********************)
	IF Event.no[1].Text2 <> Name AND Name <> '' OR Event.no[1].Text2 = '' AND rAxis.NcToPlc.AxisId <> 0
	THEN
		Event.no[1].Class 									:= TC2_SYSTEM.TCEVENTCLASS_STATEINFO;
		Event.no[3].Class 									:= TC2_SYSTEM.TCEVENTCLASS_MESSAGE;
		Event.no[4].Class 									:= TC2_SYSTEM.TCEVENTCLASS_WARNING;
		Event.no[5].Class 									:= TC2_SYSTEM.TCEVENTCLASS_STATEINFO;
		Event.no[6].Class 									:= TC2_SYSTEM.TCEVENTCLASS_STATEINFO;
		Event.no[7].Class 									:= TC2_SYSTEM.TCEVENTCLASS_STATEINFO;
		
		(* Init axisname *)
		FOR i := Event.MIN_EVENT TO Event.MAX_EVENT DO
		(*	Event.no[i].Text1								:= '';*)
			Event.no[i].Text2								:= SEL(LEN(name)>1,CONCAT('Axis id:',DWORD_TO_STRING(rAxis.NcToPlc.AxisId)),name);			
		END_FOR
		
	END_IF

(* workl Event Ctrl *************************************************)
	Event(
		ConfirmTrig 	:= ConfirmTrig,
		Disable			:= rAxis.NcToPlc.AxisId = 0 OR NOT EnableEvent,
		SourceId		:= SourceId + rAxis.NcToPlc.AxisId);
		
	NoOfActiveEvents										:= Event.NoOfActiveEvents ;
 	EventStatus												:= Event.Status ;
	
(*********************************************************************************)

END_FUNCTION_BLOCK

// POUs/IO/Drives/CoE/InovanceSV660/CiA_DS402Statusword_INOVANCE
FUNCTION_BLOCK CiA_DS402Statusword_INOVANCE EXTENDS CiA_DS402Statusword
VAR_INPUT
END_VAR
VAR_OUTPUT	
	TargetReached			: BOOL; // Bit 10 commonly used for in target position, velocity ect.
	HomeFound				: BOOL; // Bit 15: 
END_VAR

METHOD PUBLIC readStatusword : BOOL
VAR_INPUT
	Statusword 		:	UINT;
END_VAR
SUPER^.readStatusword(Statusword);

TargetReached												:= Statusword.10;
HomeFound													:= Statusword.15;
readStatusword												:= TRUE;
END_METHOD

END_FUNCTION_BLOCK

// POUs/IO/Drives/CoE/StaeubliCS8/AxDriveCoE_StaeubliCS8
{attribute 'no_check'}
//Staeubli CS8 robot control with CoE EtherCAT interface  
//EventHandling instance use inside
FUNCTION_BLOCK AxDriveCoE_StaeubliCS8 EXTENDS AxDriveBase                         						
VAR_INPUT                           						
	EnableEvent												:	BOOL := TRUE;
	ConfirmTrig												:	BOOL := FALSE; (* Reset event Flag *)
	SourceId												:	UDINT := 102200; //CoE Drive default multisource Id + Ax id
	Name													:	STRING(30) := '';
	ErrorLimitPos											:	BOOL := FALSE;
	ErrorLimitNeg											:	BOOL := FALSE;
END_VAR
VAR_IN_OUT
END_VAR
VAR_OUTPUT
	LiveCountTimeout										:	BOOL;
	LiveCount										AT %I* 	:	USINT;	(* Wenn diese Variable nicht vorhanden ist bitte mit NCtoPLC *)
	CanNodeState									AT %I* 	:	USINT; (* Master- AND Slave-Mode:
   																						0 = No error
                        							
																						Master-Mode:
																						   1 = Node deactivated
																						   2 = Node not found
																						   4 = SDO syntax error at StartUp
																						   5 = SDO data mismatch at StartUp
																						   8 = Node StartUp in progress
																						  11 = FC510x Bus-OFF
																						  12 = Pre-Operational
																						  13 = Severe bus fault
																						  14 = Guarding: toggle error
																						  20 = TxPDO too short
																						  22 = Expected TxPDO is missing
																						  23 = Node is Operational but not all TxPDOs were received
																						  31 = only for EtherCAT gateways: WC-State of cyclic EtherCAT frame is 1
                        							
																						Slave-Mode:
																						 128 = Node is Operational but not all RxPDOs were received
																						 129 = Node is Pre-Operational
																						 130 = Node is Stopped *)
	Status													:	CiA_DS402Statusword_StaeubliCS8;	
	EventStatus												:	DWORD;
	NoOfActiveEvents										:	INT;
	Busy													:	BOOL;
	Error													:	BOOL;
{attribute 'displaymode':='hex'}
	ErrorId													:	UDINT;
END_VAR                             						
VAR

END_VAR
VAR

(* Cache *********************************************************************)
	MemLiveCount											:	USINT;
	
(* Timer ********************************************************************************)
	TON_LiveCountTimeout									:	TON;
	TON_NotEnabled											:	TON;
                                    						
(* Trigger ******************************************************************************)

(* Bausteine ****************************************************************************)
	Event													:	EventHandlingGrp25;

(* Dummy Speicher **********************************************************)
	i														:	INT;
(****************************************************************************)
END_VAR

	(* CS8 Staeubli Robot Control as Ethercat Slave Drive 								*)
	(************************************************************************************)

(* abort function-call if the reference is invalid *****************************)
IF NOT __ISVALIDREF(rAxis) 
THEN
	Busy													:= NOT Error;
	Fault													:= TRUE;
	SwitchedOn												:= FALSE;
	Ready													:= FALSE;
	Error													:= TRUE;
	ErrorId													:= 16#4B30;
	RETURN;         										
END_IF

(* Read Statusword ********************************************************)
	(* LiveCount Timeout ************************************)
	TON_LiveCountTimeout(
		IN := MemLiveCount = LiveCount AND NOT rAxis.Status.OpMode.SimulationAxis,
		PT := t#1s,
		Q	=> LiveCountTimeout);
	
	(* DriveStatusword *****************************)
	IF LiveCountTimeout 
	THEN 
		Status.readStatusword(0);
	ELSE	
		IF rAxis.Status.OpMode.SimulationAxis
		THEN
			IF rAxis.PlcToNc.ControlDWord.0
			THEN
				Status.readStatusword(TO_UINT(eCiA_DS402_STATUS_STATE.OPERATION_ENABLED) OR 2#0100_0000_0000_0000);
			ELSE
				Status.readStatusword(TO_UINT(eCiA_DS402_STATUS_STATE.SWITCHED_ON) OR 2#0100_0000_0000_0000);	
			END_IF
		ELSE
			Status.readStatusword(Statusword);
		END_IF		
	END_IF

																															
	(*
	Bits 	Value 	Description
	15		 X 		Reserved
	14 	0/1 		Status OF position feedback value.  1: the robot axis is calibrated.  0: the robot axis is NOT calibrated.
	13 	0/1 		No following error /Following error
	12 	0/1 		Follwing command value
	11 	0/1 		Internal LIMIT active
	10 	0/1		Target reached
	9 		0/1 		Remote
	8 		0/1 		Manufacturer specific
	7 		0/1 		Warning
	6 		0/1 		Switch on disabled
	5 		1 			Quick stop. NS
	4 		0/1 		Voltage enable
	3 		0/1 		Fault
	2 		0/1 		Operation enabled
	1 		0/1 		Switched on
	0 		0/1 		Ready TO switch on
	*)

(* DriveStatusBits ***********************************************)
	Fault													:= Status.Fault
																OR Status.FollowingError
																OR NOT Status.Calibrated(* Nur bei Absolut Encoder Achsen *)
																OR rAxis.NcToPlc.StateDWord.28 (* DriveDeviceError *)
																OR rAxis.NcToPlc.StateDWord.30; (* IODataInvalid *)
            												
	Ready 													:= NOT Fault
																AND(Status.ReadyToSwitchOn OR Status.SwitchedOn);

	SwitchedOn												:= Status.SwitchedOn AND NOT Fault AND(Status.FollowCmdValue OR Status.RemoteActive);
	
(* Event Logger Meldungen *****************************************************)
	TON_NotEnabled(
		IN := Status.SwitchedOn AND NOT Status.OperationEnabled AND Ready,
		PT := t#2s);

	Event.no[1].Flag 										:= NOT Status.ReadyToSwitchOn; 
	Event.no[2].Flag 										:= Status.Fault;
	Event.no[3].Flag 										:= Status.Warning; 				
	Event.no[4].Flag 										:= Status.InternalLimitActive;
	Event.no[5].Flag 										:= Status.SwitchOnDisabled;
	Event.no[6].Flag 										:= NOT Status.FollowCmdValue AND Status.SwitchedOn AND NOT rAxis.Status.OpMode.SimulationAxis;		
	Event.no[7].Flag 										:= FALSE;									
	Event.no[8].Flag 										:= ErrorLimitPos;
	Event.no[9].Flag 										:= ErrorLimitNeg;
	Event.no[10].Flag 										:= FALSE;
	
	Event.no[11].Flag 										:= NOT Status.RemoteActive;
	Event.no[12].Flag 										:= Status.FollowingError ;	
	Event.no[13].Flag 										:= NOT Status.Calibrated ; 	(* Nur bei Absolut Encoder Achsen *)
	Event.no[14].Flag 										:= CanNodeSTATE = 128; 					(* Node is Operational but not all RxPDOs were received *)
	Event.no[15].Flag 										:= CanNodeSTATE = 129; 					(* Node is Pre-Operational *)
	Event.no[16].Flag 										:= CanNodeSTATE = 130;					(* Node is Stopped *)
	Event.no[17].Flag 										:= TON_NotEnabled.Q; 			
	Event.no[18].Flag 										:= LiveCountTimeout ; 			
(*	Event.no[19].Flag 										:= FALSE;
	Event.no[20].Flag 										:= FALSE;
	Event.no[21].Flag 										:= FALSE;
	Event.no[22].Flag 										:= FALSE;
	Event.no[23].Flag 										:= FALSE;
	Event.no[24].Flag 										:= FALSE;
	Event.no[25].Flag 										:= FALSE; *)

(* Check if msg activ and init some parameter ***********************)
	IF Event.no[1].Text2 <> Name AND Name <> '' OR Event.no[1].Text2 = '' AND rAxis.NcToPlc.AxisId <> 0
	THEN
		Event.no[1].Class 									:= TC2_SYSTEM.TCEVENTCLASS_STATEINFO;
		Event.no[3].Class 									:= TC2_SYSTEM.TCEVENTCLASS_WARNING;
		Event.no[4].Class 									:= TC2_SYSTEM.TCEVENTCLASS_WARNING;
		Event.no[5].Class 									:= TC2_SYSTEM.TCEVENTCLASS_STATEINFO;
		Event.no[6].Class 									:= TC2_SYSTEM.TCEVENTCLASS_STATEINFO;

		Event.no[11].Class 									:= TC2_SYSTEM.TCEVENTCLASS_STATEINFO;
		Event.no[17].Class 									:= TC2_SYSTEM.TCEVENTCLASS_WARNING;
		Event.no[18].Class 									:= TC2_SYSTEM.TCEVENTCLASS_WARNING;
		
		(* Init axisname *)
		FOR i := Event.MIN_EVENT TO Event.MAX_EVENT DO
		(*	Event.no[i].Text1								:= '';*)
			Event.no[i].Text2								:= SEL(LEN(name)>1,CONCAT('Axis id:',DWORD_TO_STRING(rAxis.NcToPlc.AxisId)),name);
		END_FOR
	END_IF

(* workl Event Ctrl *************************************************)
	Event(
		ConfirmTrig 	:= ConfirmTrig,
		Disable			:= rAxis.NcToPlc.AxisId = 0 OR NOT EnableEvent,
		SourceId		:= SourceId + rAxis.NcToPlc.AxisId,
		Status			=> EventStatus,
		NoOfActiveEvents => NoOfActiveEvents);

(******************************************************************************)

METHOD PUBLIC confirm : bool
VAR_INPUT
END_VAR
confirm								:= Event.confirm();
END_METHOD

END_FUNCTION_BLOCK

// POUs/IO/Drives/CoE/StaeubliCS8/CiA_DS402Statusword_StaeubliCS8
FUNCTION_BLOCK CiA_DS402Statusword_StaeubliCS8 EXTENDS CiA_DS402Statusword
VAR_INPUT
END_VAR
VAR_OUTPUT	
	FollowingError			: BOOL; // Bit 13: Following error occured
	Calibrated				: BOOL; // Bit 14: Motor calibrated
END_VAR

METHOD PUBLIC readStatusword : BOOL
VAR_INPUT
	Statusword 		:	UINT;

END_VAR

FollowingError												:= Statusword.13 ;
Calibrated													:= Statusword.14 ;

readStatusword												:= SUPER^.readStatusword(Statusword);
END_METHOD

END_FUNCTION_BLOCK
